{attribute addProperty BoxType "EKM1101-0000-0016"}
{attribute addProperty Id "TimestampAT %I*ULINT648"}
{attribute addProperty CRC "187023780"}
{attribute addProperty SizeInBites "64"}
{attribute addProperty SizeInBytes "8"}
TYPE MMS_Acceleration_Timestamp_0B25C1A4 :
STRUCT
	{attribute addProperty Name "Timestamp"}
	Timestamp AT %I* : ULINT;
END_STRUCT
END_TYPE

(* stored: Version 1.2.0.0, ProductVersion 3.1.4024.9
   DUT MMS_Acceleration_Timestamp_0B25C1A4: Id {4a9d6684-4024-44c8-88ef-310f5eeab91c} *)
